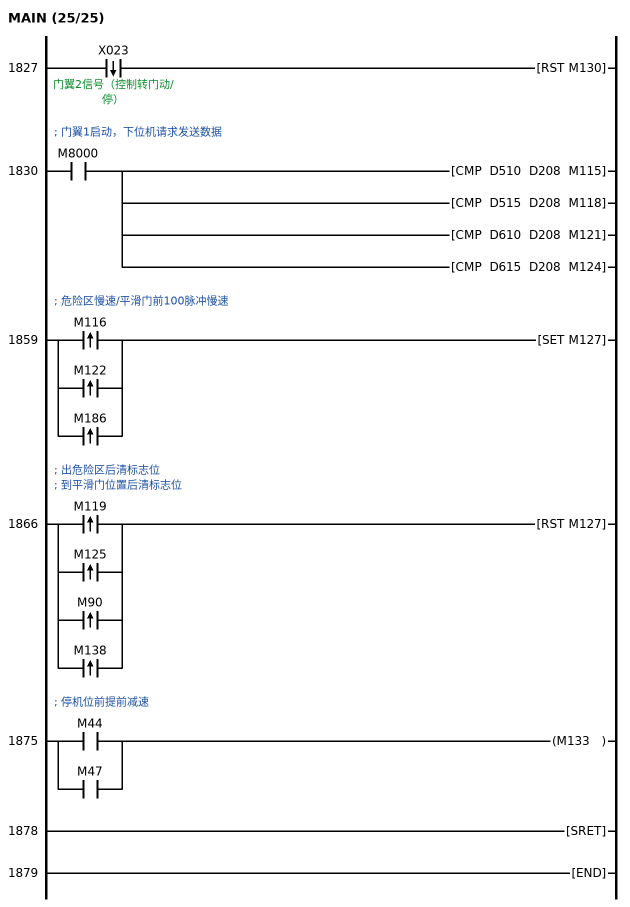
[picture p24: ladder of MAIN, rungs at steps 1827 to 1879]
1827  LDF     X023  ; 门翼2信号（控制转门动/停）
      RST     M130
        [note] 第二个门翼关好后：M130=0
; 门翼1启动，下位机请求发送数据
1830  LD      M8000
      CMP     D510 D208 M115
        [note] 危险区1起点位置：M116=1
      CMP     D515 D208 M118
        [note] 危险区1终点位置：M119=1
      CMP     D610 D208 M121
        [note] 危险区2起点位置：M122=1
      CMP     D615 D208 M124
        [note] 危险区2终点位置：M125=1
; 危险区慢速/平滑门前100脉冲慢速
1859  LDP     M116
      ORP     M122
      ORP     M186
      SET     M127
        [note] 到危险区时慢速：Y1+Y7
; 出危险区后清标志位
; 到平滑门位置后清标志位
1866  LDP     M119
      ORP     M125
      ORP     M90
      ORP     M138
      RST     M127
        [note] 出危险区后恢复
; 停机位前提前减速
1875  LD      M44
      OR      M47
      OUT     M133
        [note] 慢速--Y6
1878  SRET
1879  END
END_PROGRAM
